{attribute 'qualified_only'}
VAR_GLOBAL
B1: BOOL; 		// Lichtschranke draussen
B2:	BOOL; 		//Lichtschranke drinnen 
Auto: BYTE; 	//Anzahl Autos
Personen: BYTE; // Anzahl Personen
END_VAR

(* stored: Version 1.1.0.1, ProductVersion 3.1.4022.7
   GVL ADS: Id {1151171f-0ef3-4d6c-9971-70afc555383b} *)
